# B&R Automation Studio project GAT (part 10)

### mappFrameworkGlobal.var - not listed in the package file held
```iecst
VAR
	gbUSBAvail : ARRAY[0..MAX_IDX_USB_DEV_LIST] OF BOOL; (*Status array of USB storage devices*)
END_VAR
```

Listed in the project but not available here: Logical/Infrastructure/AlarmX/AlarmMgr/AlarmHandling.st, Logical/Infrastructure/Audit/AuditMgr/AuditMgt.typ, Logical/Infrastructure/Audit/AuditMgr/AuditMgt.var, Logical/Infrastructure/Data/DataMgr/DataMgr.typ, Logical/Infrastructure/Data/DataMgt/DataMgt.typ, Logical/Infrastructure/File/File/FileMgt.typ, Logical/Infrastructure/File/File/FileMgt.var, Logical/Infrastructure/Recipe/Recipe/Recipe.var, Logical/Infrastructure/Recipe/Recipe/HMIActions.st, Logical/Infrastructure/UserX/UserXMgr/UserXMgr.typ, Logical/Infrastructure/UserX/UserXMgt/UserX.typ, Logical/Infrastructure/UserX/UserXMgt/UserX.fun, Logical/Infrastructure/TS_UnitTest/Samples/Framework_Extension_With_Custom_Asserts/LibAssert1/LibAssert1.h, Logical/Infrastructure/TS_UnitTest/Samples/Framework_Extension_With_Custom_Asserts/LibAssert1/LibAssert1_ThresholdAssert.h, Logical/Infrastructure/TS_UnitTest/Samples/Framework_Extension_With_Custom_Asserts/LibAssert1/LibAssert1_ThresholdAssert.c, Logical/Infrastructure/TS_UnitTest/Samples/Framework_Extension_With_Custom_Asserts/LibAssert1/LibAssert1_REAL_ArrayAsserts.h, Logical/Infrastructure/TS_UnitTest/Samples/Framework_Extension_With_Custom_Asserts/LibAssert1/LibAssert1_REAL_ArrayAsserts.c, Logical/Infrastructure/TS_UnitTest/Samples/Framework_Features/SPL_Asserts/testSuite.c, Logical/Infrastructure/TS_UnitTest/Samples/Framework_Features/SPL_Asserts/autoGeneratedFile.c, Logical/Infrastructure/TS_UnitTest/Samples/Framework_Features/SPL_Asserts/varAsserts.var, Logical/Infrastructure/TS_UnitTest/Samples/Framework_Features/SPL_Asserts/testSet_Asserts.c, Logical/Infrastructure/TS_UnitTest/Samples/Framework_Features/SPL_Behavior/testSuite.var, Logical/Infrastructure/TS_UnitTest/Samples/Framework_Features/SPL_Behavior/testSuite.c, Logical/Infrastructure/TS_UnitTest/Samples/Framework_Features/SPL_Behavior/autoGeneratedFile.c, Logical/Infrastructure/TS_UnitTest/Samples/Framework_Features/SPL_Behavior/iPrototypes.h, Logical/Infrastructure/TS_UnitTest/Samples/Framework_Features/SPL_Behavior/iHelperFunction.h, Logical/Infrastructure/TS_UnitTest/Samples/Framework_Features/SPL_Behavior/iHelperFunction.c, Logical/Infrastructure/TS_UnitTest/Samples/Framework_Features/SPL_Behavior/TestBusy_AsyncronousVariables.var, Logical/Infrastructure/TS_UnitTest/Samples/Framework_Features/SPL_Behavior/TestBusy_Asyncronous, Logical/Infrastructure/TS_UnitTest/Templates/HelperTool_Supported/utTemplate_automated/variables.var, Logical/Infrastructure/TS_UnitTest/Templates/NoToolSupport/utTemplate_manual/variables.var, Logical/Infrastructure/TS_UnitTest/Templates/NoToolSupport/utTemplate_manual/testSuite.c, Logical/Infrastructure/TS_UnitTest/Templates/NoToolSupport/utTemplate_manual/FixtureOfTestSets.c, Logical/Infrastructure/AxisTemplate/AxisMgr/AxisMgr.st, Logical/Infrastructure/AxisTemplate/AxisMgr/AxisMgr.typ, Logical/Infrastructure/AxisTemplate/AxisMgr/AxisMgr.var, Logical/Infrastructure/AxisTemplate/AxisMgr/Variables.var, Logical/Infrastructure/AxisTemplate/AxisMgr/AxisStateMachine.st, Logical/Infrastructure/AxisTemplate/AxisMgr/AxisControlModes.st, Logical/Infrastructure/AxisTemplate/AxisMgr/Recipe.st, Logical/Infrastructure/AxisTemplate/AxisMgr/SimulationControl.st, Logical/Infrastructure/AxisTemplate/AxisMgr/LocalFunctions.fun, Logical/Infrastructure/AxisTemplate/AxisMgr/ManualCommand.st, Logical/Infrastructure/AxisTemplate/AxisMgr/AutomaticCommand.st, Logical/Infrastructure/AxisTemplate/AxisMgr/ChangeConfiguration.st, Logical/Infrastructure/AxisTemplate/UnitTests/prototypeTest/TestType.typ, Logical/Infrastructure/AxisTemplate/UnitTests/prototypeTest/Set_SetupTeardown.c, Logical/Infrastructure/AxisTemplate/UnitTests/prototypeTest/autoGeneratedFile.c, Logical/Infrastructure/AxisTemplate/AxisMgr/AxisMgr.typ, Logical/Infrastructure/AxisTemplate/AxisControl/LocalFunctions.fun, Logical/Infrastructure/UsbDevLink/UsbDevLink/UsbDevLink.typ, Logical/MachineControl/AxisTemplate/UnitTests/prototypeTest/TestType.typ, Logical/MachineControl/AxisTemplate/UnitTests/prototypeTest/variables.var, Logical/MachineControl/AxisTemplate/UnitTests/prototypeTest/testSuite.c, Logical/MachineControl/AxisTemplate/UnitTests/prototypeTest/Set_SetupTeardown.c, Logical/MachineControl/AxisTemplate/UnitTests/prototypeTest/autoGeneratedFile.c, Logical/MachineControl/AppAxis_1/AppAxis_1/AxisMgr.st, Logical/MachineControl/AppAxis_1/AppAxis_1/Variables.var, Logical/MachineControl/AxisTemplate/AxisMgr/AxisStateMachine.st, Logical/MachineControl/AppAxis_1/AppAxis_1/ManualCommand.st, Logical/MachineControl/AxisTemplate/AxisMgr/ChangeConfiguration.st, Logical/MachineControl/CrossCutter/CrossCutter/AxisControl.typ, Logical/MachineControl/CrossCutter/CrossCutter/Variables.var, Logical/MachineControl/CrossCutter/CrossCutter/LocalFunctions.fun, Logical/Infrastructure/AxisTemplate/AxisMgr/AxisMgr.var, Logical/Infrastructure/AxisTemplate/AxisMgr/AxisStateMachine.st, Logical/Infrastructure/AxisTemplate/AxisMgr/ChangeConfiguration.st, Logical/Infrastructure/AxisTemplate/AxisMgr/Recipe.st, Logical/MachineControl/CrossCutter/UnitTests/CutterTest/TestType.typ, Logical/MachineControl/CrossCutter/UnitTests/CutterTest/variables.var, Logical/MachineControl/CrossCutter/UnitTests/CutterTest/testSuite.c, Logical/MachineControl/CrossCutter/UnitTests/CutterTest/Set_SetupTeardown.c, Logical/MachineControl/CrossCutter/UnitTests/CutterTest/autoGeneratedFile.c, Logical/MachineControl/CrossCutter/CrossCutter/AxisControl.typ, Logical/MachineControl/Conveyor/Conveyor/Variables.var, Logical/MachineControl/Conveyor/Conveyor/LocalFunctions.fun, Logical/MachineControl/Conveyor/Conveyor/ManualCommand.st, Logical/MachineControl/Conveyor/UnitTests/ConvTest/TestType.typ, Logical/MachineControl/Conveyor/UnitTests/ConvTest/variables.var, Logical/MachineControl/Conveyor/UnitTests/ConvTest/testSuite.c, Logical/MachineControl/Conveyor/UnitTests/ConvTest/Set_SetupTeardown.c, Logical/MachineControl/Conveyor/UnitTests/ConvTest/autoGeneratedFile.c, Logical/ChineseHelp, Logical/UserPartition/Audit, Logical/UserPartition/Data, Logical/UserPartition/Report
